{attribute 'call_after_init'}
FUNCTION_BLOCK FB_BaseplateChillerEnable_Test EXTENDS FB_TestSuite
VAR_INPUT
END_VAR
VAR_OUTPUT
END_VAR
VAR
END_VAR

LocksWithHardwareFailure();
LocksWithLUTLeak();
EnablesWhenNoError();

METHOD EnablesWhenNoError
VAR
	stErrors : st_ErrorStates;
	bResult : BOOL;
END_VAR
TEST('EnablesWhenNoError');

bResult := F_BaseplateChillerEnable(stErrors := stErrors);

AssertTrue(bResult, 'Baseplate chiller relay did not close');

TEST_FINISHED();
END_METHOD

METHOD LocksWithHardwareFailure
VAR
	stErrors : st_ErrorStates;
	bResult : BOOL;
END_VAR
TEST('LocksWithHardwareFailure');

stErrors.bHardwareFailure := TRUE;
bResult := F_BaseplateChillerEnable(stErrors := stErrors);

AssertFalse(bResult, 'Baseplate chiller relay did not open');

TEST_FINISHED();
END_METHOD

METHOD LocksWithLUTLeak
VAR
	stErrors : st_ErrorStates;
	bResult : BOOL;
END_VAR
TEST('LocksWithLUTLeak');

stErrors.bLeakUnderTable := TRUE;
bResult := F_BaseplateChillerEnable(stErrors := stErrors);

AssertFalse(bResult, 'Baseplate chiller relay did not open');

TEST_FINISHED();
END_METHOD

END_FUNCTION_BLOCK

(* stored: Version 1.1.0.1, ProductVersion 3.1.4022.17
   POU FB_BaseplateChillerEnable_Test: Id {1f6e178b-ccad-4d1a-b854-05819cec5772}, SpecialFunc None
   Method EnablesWhenNoError: Id {57f6cef7-3faf-4ddd-a400-3eedade2fa36}
   Method LocksWithHardwareFailure: Id {0f653f74-9cd9-48f3-952e-e731656590da}
   Method LocksWithLUTLeak: Id {0c1ef9cd-1633-45b8-9e32-826a019b837e} *)
